// TwinCAT 3 PLC project Main
// ProgramVersion: 3.1.4024.0
// libraries:
//   Tc2_Standard, * (Beckhoff Automation GmbH)
//   Tc2_System, * (Beckhoff Automation GmbH)
//   Tc3_Module, * (Beckhoff Automation GmbH)
//   TcUnit, * (www.tcunit.org)
//   [mobject-promises], * (mobject)
// project tree:
//   Programs/ Main.TcPOU
//   Tasks/ PlcTask.TcTTO
//   Tests/ Promise_TestSuite.TcPOU
// real-time tasks:
//   TASK PlcTask: cycle T#10ms, priority 20, ADS port 350

CONFIGURATION Main
    RESOURCE PLC ON TwinCAT3
        TASK PlcTask(INTERVAL := T#10ms, PRIORITY := 20);
        PROGRAM Main WITH PlcTask : Main;
    END_RESOURCE
END_CONFIGURATION

// ---- Programs/Main.TcPOU
PROGRAM Main
VAR
	promise_TestSuite : Promise_TestSuite;
END_VAR

TcUnit.Run();

END_PROGRAM

// ---- Tests/Promise_TestSuite.TcPOU
FUNCTION_BLOCK Promise_TestSuite EXTENDS TcUnit.FB_TestSuite
VAR
END_VAR

TestPromisePending();
TestPromiseReject();
TestPromiseResolve();
TestPromiseTryGetEntity();
TestPromiseTryGetEntityTo();
TestPromiseTryGetResult();
TestPromiseTryGetResultTo();
TestPromiseTrySetEntity();

METHOD TestPromisePending
VAR
	promise : Promise;
	pendingResult : BOOL;
	resolvedResult : BOOL;
	rejectedResult : BOOL;
	rejectedReason : T_MAXSTRING;
	expectedReson : T_MAXSTRING := '';
END_VAR
TEST('TestPromisePending');

pendingResult := promise.Pending;
resolvedResult := promise.Resolved;
rejectedResult := promise.Rejected;
rejectedReason := promise.RejectedReason;

AssertTrue(
	Condition := pendingResult,
	Message := 'Incorrect state of Pending'
);

AssertFalse(
	Condition := resolvedResult,
	Message := 'Incorrect state of Resolved'
);

AssertFalse(
	Condition := rejectedResult,
	Message := 'Incorrect state of Rejected'
);

AssertEquals(
	Expected := expectedReson,
	Actual := rejectedReason,
	Message := 'Incorrect reject reason'
);

TEST_FINISHED();
END_METHOD

METHOD TestPromiseReject
VAR
	promise : Promise;
	pendingResult : BOOL;
	resolvedResult : BOOL;
	rejectedResult : BOOL;
	rejectedReason : T_MAXSTRING;
	expectedReson : T_MAXSTRING := 'test message';
END_VAR
TEST('TestPromiseReject');

promise.Ctx.Reject('test message');

pendingResult := promise.Pending;
resolvedResult := promise.Resolved;
rejectedResult := promise.Rejected;
rejectedReason := promise.RejectedReason;

AssertFalse(
	Condition := pendingResult,
	Message := 'Incorrect state of Pending'
);

AssertFalse(
	Condition := resolvedResult,
	Message := 'Incorrect state of Resolved'
);

AssertTrue(
	Condition := rejectedResult,
	Message := 'Incorrect state of Rejected'
);

AssertEquals(
	Expected := expectedReson,
	Actual := rejectedReason,
	Message := 'Incorrect reject reason'
);

TEST_FINISHED();
END_METHOD

METHOD TestPromiseResolve
VAR
	promise : Promise;
	pendingResult : BOOL;
	resolvedResult : BOOL;
	rejectedResult : BOOL;
	rejectedReason : T_MAXSTRING;
	expectedReson : T_MAXSTRING := '';
END_VAR
TEST('TestPromiseResolve');

promise.Ctx.Resolve();

pendingResult := promise.Pending;
resolvedResult := promise.Resolved;
rejectedResult := promise.Rejected;
rejectedReason := promise.RejectedReason;

AssertFalse(
	Condition := pendingResult,
	Message := 'Incorrect state of Pending'
);

AssertTrue(
	Condition := resolvedResult,
	Message := 'Incorrect state of Resolved'
);

AssertFalse(
	Condition := rejectedResult,
	Message := 'Incorrect state of Rejected'
);

AssertEquals(
	Expected := expectedReson,
	Actual := rejectedReason,
	Message := 'Incorrect reject reason'
);

TEST_FINISHED();
END_METHOD

METHOD TestPromiseTryGetEntity
VAR
	promise : Promise;
	value : T_MAXSTRING := 'myTest';
	getResult : BOOL;
	actualResult : T_MAXSTRING;
	expectedResult : T_MAXSTRING := 'myTest';
END_VAR
TEST('TestPromiseTryGetEntity');

promise.Ctx.TrySetEntity('myString',value);
getResult := promise.Ctx.TryGetEntity('myString',actualResult);

AssertTrue(
	Condition := getResult,
	Message := 'Unable to return the context entity'
);

AssertEquals(
	Expected := actualResult,
	Actual := expectedResult,
	Message := 'Incorrect returned entity from the context'
);

TEST_FINISHED();
END_METHOD

METHOD TestPromiseTryGetEntityTo
VAR
	promise : Promise;
	value : T_MAXSTRING := 'myTest';
	getResult : BOOL;
	actualResult : T_MAXSTRING;
	expectedResult : T_MAXSTRING := 'myTest';
END_VAR
TEST('TestPromiseTryGetEntityTo');

promise.Ctx.TrySetEntity('myString',value);
getResult := promise.Ctx.TryGetEntityTo('myString',ADR(actualResult),SIZEOF(actualResult));

AssertTrue(
	Condition := getResult,
	Message := 'Unable to return the context entity'
);

AssertEquals(
	Expected := actualResult,
	Actual := expectedResult,
	Message := 'Incorrect returned entity from the context'
);

TEST_FINISHED();
END_METHOD

METHOD TestPromiseTryGetResult
VAR
	promise : Promise;
	value : INT := 123;
	pendingResult : BOOL;
	resolvedResult : BOOL;
	rejectedResult : BOOL;
	rejectedReason : T_MAXSTRING;
	expectedReson : T_MAXSTRING := '';
	tryGetResult : BOOL;
	actualResult : INT;
	expectedResult : INT := 123;
END_VAR
TEST('TestPromiseTryGetResult');

promise.Ctx.ResolveWith(value);

pendingResult := promise.Pending;
resolvedResult := promise.Resolved;
rejectedResult := promise.Rejected;
rejectedReason := promise.RejectedReason;

tryGetResult := promise.TryGetResult(actualResult);

AssertFalse(
	Condition := pendingResult,
	Message := 'Incorrect state of Pending'
);

AssertTrue(
	Condition := resolvedResult,
	Message := 'Incorrect state of Resolved'
);

AssertFalse(
	Condition := rejectedResult,
	Message := 'Incorrect state of Rejected'
);

AssertTrue(
	Condition := tryGetResult,
	Message := 'Unable to get result'
);

AssertEquals(
	Expected := expectedReson,
	Actual := rejectedReason,
	Message := 'Incorrect reject reason'
);

AssertEquals(
	Expected := actualResult,
	Actual := expectedResult,
	Message := 'Incorrect returned result'
);

TEST_FINISHED();
END_METHOD

METHOD TestPromiseTryGetResultTo
VAR
	promise : Promise;
	value : INT := 123;
	pendingResult : BOOL;
	resolvedResult : BOOL;
	rejectedResult : BOOL;
	rejectedReason : T_MAXSTRING;
	expectedReson : T_MAXSTRING := '';
	tryGetResult : BOOL;
	actualResult : INT;
	expectedResult : INT := 123;
END_VAR
TEST('TestPromiseTryGetResultTo');

promise.Ctx.ResolveWith(value);

pendingResult := promise.Pending;
resolvedResult := promise.Resolved;
rejectedResult := promise.Rejected;
rejectedReason := promise.RejectedReason;

tryGetResult := promise.TryGetResultTo(ADR(actualResult),SIZEOF(actualResult));

AssertFalse(
	Condition := pendingResult,
	Message := 'Incorrect state of Pending'
);

AssertTrue(
	Condition := resolvedResult,
	Message := 'Incorrect state of Resolved'
);

AssertFalse(
	Condition := rejectedResult,
	Message := 'Incorrect state of Rejected'
);

AssertTrue(
	Condition := tryGetResult,
	Message := 'Unable to get result'
);

AssertEquals(
	Expected := expectedReson,
	Actual := rejectedReason,
	Message := 'Incorrect reject reason'
);

AssertEquals(
	Expected := actualResult,
	Actual := expectedResult,
	Message := 'Incorrect returned result'
);

TEST_FINISHED();
END_METHOD

METHOD TestPromiseTrySetEntity
VAR
	promise : Promise;
	value : INT := 123;
	actualResult : INT;
	expectedResult : INT := 123;
END_VAR
TEST('TestPromiseTrySetEntity');

promise.Ctx.TrySetEntity('myNumber',value);
promise.Ctx.TryGetEntity('myNumber',actualResult);

AssertEquals(
	Expected := actualResult,
	Actual := expectedResult,
	Message := 'Incorrect returned entity from the context'
);

TEST_FINISHED();
END_METHOD

END_FUNCTION_BLOCK
